PROGRAM SFC
VAR
	count : INT := 0;
	reset : BOOL := FALSE;
END_VAR

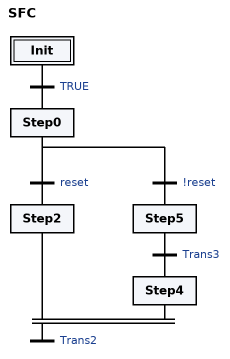
INITIAL_STEP Init:
END_STEP
TRANSITION FROM Init TO Step0
    := TRUE;
END_TRANSITION
STEP Step0:
END_STEP
TRANSITION FROM Step0 TO Step2
    := reset;
END_TRANSITION
STEP Step2:
END_STEP
TRANSITION FROM Step0 TO Step5
    := !reset;
END_TRANSITION
STEP Step5:
END_STEP
TRANSITION FROM Step5 TO Step4
    := Trans3;
END_TRANSITION
STEP Step4:
END_STEP
TRANSITION FROM (Step2, Step4) TO ???
    := Trans2;
END_TRANSITION

ACTION Step5_entry:
count := count + 1;
END_ACTION

END_PROGRAM

(* stored: Version 1.1.0.1, ProductVersion 3.1.4024.12
   POU SFC: Id {301fa998-fba7-42e4-9e73-18b507c3cbce}, SpecialFunc None
   Action Step5_entry: Id {99a20b9b-5303-4659-b1ef-70f0d870c7fe} *)
